FUNCTION_BLOCK AnalogOutput EXTENDS Component IMPLEMENTS I_AnalogOutput, I_AnalogScalable, I_CalibratableLinear
VAR
	Output			 : REFERENCE TO INT;
	Forcible		 : ForcibleInt(_Name);
	_Scale			 : I_AnalogScale;
	_CalibrateLinear : I_CalibrateLinear;
	_CalibrateCustom : I_TransformLRealValue;
END_VAR

VAR
	{attribute 'hide'}
	DefaultScale : AnalogScale;
	{attribute 'hide'}
	DefaultCalibration : Calibrate;
END_VAR

PROPERTY CalibrateCustom : I_TransformLrealValue
SET
_CalibrateCustom := CalibrateCustom;
END_SET
END_PROPERTY

PROPERTY CalibrateLinear : I_CalibrateLinear
GET
CalibrateLinear := _CalibrateLinear;
END_GET
SET
_CalibrateLinear := CalibrateLinear;
END_SET
END_PROPERTY

(*FB_Init is always available implicitly and it is used primarily for initialization.
The return value is not evaluated. For a specific influence, you can also declare the
methods explicitly and provide additional code there with the standard initialization
code. You can evaluate the return value.*)
METHOD FB_Init : BOOL
VAR_INPUT
	(* TRUE: the retain variables are initialized (reset warm / reset cold)*)
	bInitRetains : BOOL;

	(* TRUE: the instance will be copied to the copy code afterward (online change)   *)
	bInCopyCode : BOOL;
	Name		: T_MaxString;
	Output		: REFERENCE TO INT;
END_VAR
_Scale			 := DefaultScale;
_CalibrateLinear := DefaultCalibration;
THIS^.Output	 REF= Output;
END_METHOD

{attribute 'monitoring' := 'call'}
PROPERTY Force : E_ForceState
GET
Force := Forcible.CurrentForceState;
END_GET
SET
VAR
	ForceString : T_MaxString := TO_STRING(Force);
END_VAR
Forcible.SetForceState(Force);
END_SET
END_PROPERTY

PROPERTY ForceValue : INT
GET
ForceValue := Forcible.ForceValue;
END_GET
SET
Forcible.ForceValue := ForceValue;
END_SET
END_PROPERTY

{attribute 'monitoring' := 'call'}
PROPERTY RawValue : INT
GET
RawValue := Output;
END_GET
SET
Forcible.Input := RawValue;
Output		   := Forcible.Output;
END_SET
END_PROPERTY

PROPERTY Scale : I_AnalogScale
GET
Scale := _Scale;
END_GET
SET
_Scale := Scale;
END_SET
END_PROPERTY

{attribute 'monitoring' := 'call'}
PROPERTY Value : LREAL
GET
IF _CalibrateCustom = 0 THEN
	Value := _CalibrateLinear.Transform(_Scale.Transform(RawValue));
ELSE
	Value := _CalibrateCustom.Transform(_Scale.Transform(RawValue));
END_IF
END_GET
SET
IF _CalibrateCustom = 0 THEN
	RawValue := LREAL_TO_INT(_Scale.Transform(_CalibrateLinear.Transform(Value, TRUE)));
ELSE
	RawValue := LREAL_TO_INT(_Scale.Transform(_CalibrateCustom.Transform(Value, TRUE)));
END_IF
END_SET
END_PROPERTY

END_FUNCTION_BLOCK

(* stored: Version 1.1.0.1, ProductVersion 3.1.4026.18
   POU AnalogOutput: Id {7ac7b465-3ea6-4a4b-a148-c7c7ca366b31}, SpecialFunc None
   Property CalibrateCustom: Id {04dcee8b-a1cc-4f1a-836f-3d0d008232b8}
   Set Set: Id {9d385b0f-d874-4736-9ee0-aa302a5da53a}
   Property CalibrateLinear: Id {a949be51-6327-4ebe-b127-42c3188ffb68}
   Get Get: Id {c3baffc3-8374-4a90-849e-b67739613787}
   Set Set: Id {ae98b87d-60d7-46d2-9575-d6988ab4795f}
   Method FB_Init: Id {f0a06d4b-0191-43db-aa6c-266db73fd8b3}
   Property Force: Id {cefcff39-2f6d-4613-993e-9c02de9b7180}
   Get Get: Id {2393f979-99e5-4298-bc06-6835fdfe84d7}
   Set Set: Id {60605ba1-f5c7-49d8-a154-a392b3e3df4d}
   Property ForceValue: Id {a2166ad8-18ea-4e6c-8900-501742c3b4fc}
   Get Get: Id {4a64e6f6-a852-40aa-a41a-b04a29c8216b}
   Set Set: Id {5aaa7d58-59c6-4358-9012-8b157df07bd6}
   Property RawValue: Id {553d454b-200d-42b1-a096-8cb414ef4255}
   Get Get: Id {039c508d-0af9-4d11-bc75-523b85e577d3}
   Set Set: Id {0a9a00eb-b728-43a1-9b6a-04001c8b8e9a}
   Property Scale: Id {9d78ccf3-4e6e-4a17-9169-071053d01cc5}
   Get Get: Id {bdae6016-0bf2-4755-970b-6c41ede1fd4d}
   Set Set: Id {d724350c-9d4d-4e95-9b75-bd13b259a649}
   Property Value: Id {6cd4557c-222d-46fd-bea3-95d7e2d99f63}
   Get Get: Id {4cbb0c42-9e94-4e9d-85f0-da8831e13519}
   Set Set: Id {bc6b6fe3-52c1-4a9c-ba31-0596ad973380} *)
